(* PLC project Unnamed, 不明 Unnamed 1 *)
(* stored: creationDateTime 2022-12-30T13:31:29, modificationDateTime 2022-12-30T16:04:25 *)

PROGRAM prog
  VAR
    Plus : BOOL;
    Reset : BOOL;
    SetTime : TIME := T#100ms;
    Counter : INT;
    MaxValue : INT := 255;
    CTU0 : CTU;
    TON0 : TON;
    TOF0 : TOF;
  END_VAR
  VAR  (* added by the conversion: wires and edge detectors of the diagram *)
    R_TRIG1 : R_TRIG;
  END_VAR

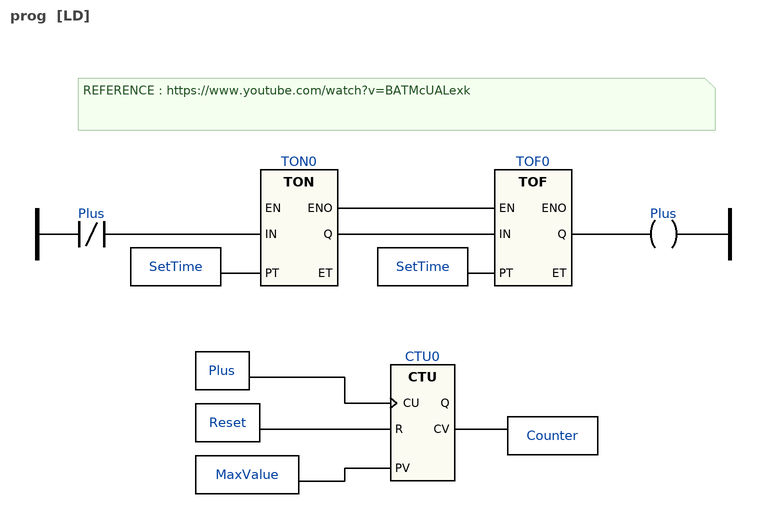
(* LD diagram, written out as Structured Text *)
(* REFERENCE : https://www.youtube.com/watch?v=BATMcUALexk *)
TON0(IN := NOT Plus, PT := SetTime);
TOF0(EN := TON0.ENO, IN := TON0.Q, PT := SetTime);
Plus := TOF0.Q;
R_TRIG1(CLK := Plus);
CTU0(CU := R_TRIG1.Q, R := Reset, PV := MaxValue);
Counter := CTU0.CV;
END_PROGRAM

CONFIGURATION Config0
  RESOURCE Res0 ON PLC
    TASK task0(INTERVAL := T#20ms, PRIORITY := 0);
    PROGRAM instance0 WITH task0 : prog;
  END_RESOURCE
END_CONFIGURATION
